{attribute 'qualified_only'}
{attribute 'strict'}
TYPE EFeedbackMsgSMD12 :
(
	PowerMsg := 10,
    InterlockStatusMsg,
    LaserTemperatureMsg,
    PsuTemperatureMsg,
    IdMsg,
    CustomMsg
);
END_TYPE

(* stored: Version 1.1.0.1, ProductVersion 3.1.4024.3
   DUT EFeedbackMsgSMD12: Id {3886e623-8368-4978-8081-7517a537689e} *)
